FUNCTION_BLOCK FB_StrategyTravelByCar IMPLEMENTS I_Strategy
VAR_INPUT
END_VAR
VAR_OUTPUT
END_VAR
VAR
END_VAR

METHOD execute
VAR_INPUT
	in_rDistance		:REAL;
END_VAR
ADSLOGSTR(msgCtrlMask:= ADSLOG_MSGTYPE_ERROR, msgFmtStr:= 'Travel time by car: %s min', strArg:= TO_STRING(in_rDistance * 0.7));
END_METHOD

END_FUNCTION_BLOCK

(* stored: Version 1.1.0.1
   POU FB_StrategyTravelByCar: Id {219046c9-c174-4b27-8de1-425c1fc405de}, SpecialFunc None
   Method execute: Id {d3fdfdee-f37e-493b-9f26-174562af75f8} *)
